FUNCTION_BLOCK SchieberControl (* Basic FB with Schieber ECC *)
  (* Standard: 61499-2; Description: Copyright (c) 2025 HR Agrartechnik GmbH This program and the accompanying materials are made available under the terms of the Eclipse Public License 2.0 which is available at https://www.eclipse.org/legal/epl-2.0/ SPDX-License-Identifier: EPL-2.0 *)
  (* Version 1.0, 2025-06-03, Franz Höpfinger, HR Agrartechnik GmbH *)
  IMPORT Schieber::AufZu::STATES;
  IMPORT Schieber::AufZu::START;
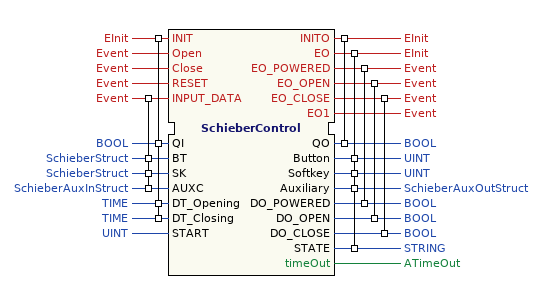
  EVENT_INPUT
    INIT : EInit WITH QI, DT_Opening, DT_Closing; (* Set all Values. Initialization Request. De-Init is not  fully supported. *)
    Open; (* Open *)
    Close; (* Close *)
    RESET; (* Reset to unknown State *)
    INPUT_DATA WITH BT, SK, AUXC;
  END_EVENT
  EVENT_OUTPUT
    INITO : EInit WITH QO; (* All Values have been Set. Initialization Confirm. *)
    EO : EInit WITH Button, Softkey, Auxiliary, STATE;
    EO_POWERED WITH DO_POWERED; (* Actuate "Open" Valve for Pneumatic *)
    EO_OPEN WITH DO_OPEN; (* Actuate "Open" Valve *)
    EO_CLOSE WITH DO_CLOSE; (* Actuate "Close" Valve *)
    EO1;
  END_EVENT
  VAR_INPUT
    QI : BOOL; (* Input event qualifier *)
    BT : SchieberStruct; (* Button *)
    SK : SchieberStruct; (* SoftKey *)
    AUXC : SchieberAuxInStruct; (* Auxiliary Control *)
    DT_Opening : TIME; (* TIME Setting *)
    DT_Closing : TIME; (* TIME Setting *)
    START : UINT := START::STARTUnknown;
  END_VAR
  VAR_OUTPUT
    QO : BOOL; (* Output event qualifier *)
    Button : UINT; (* Button Out *)
    Softkey : UINT; (* Softkey Out *)
    Auxiliary : SchieberAuxOutStruct; (* Auxiliary Control Out *)
    DO_POWERED : BOOL; (* Actuate "Open" Valve for Pneumatic *)
    DO_OPEN : BOOL; (* Actuate "Open" Valve *)
    DO_CLOSE : BOOL; (* Actuate "Close" Valve *)
    STATE : STRING;
  END_VAR
  PLUGS
    timeOut : ATimeOut; (* timeOut Adapter *)
  END_PLUGS
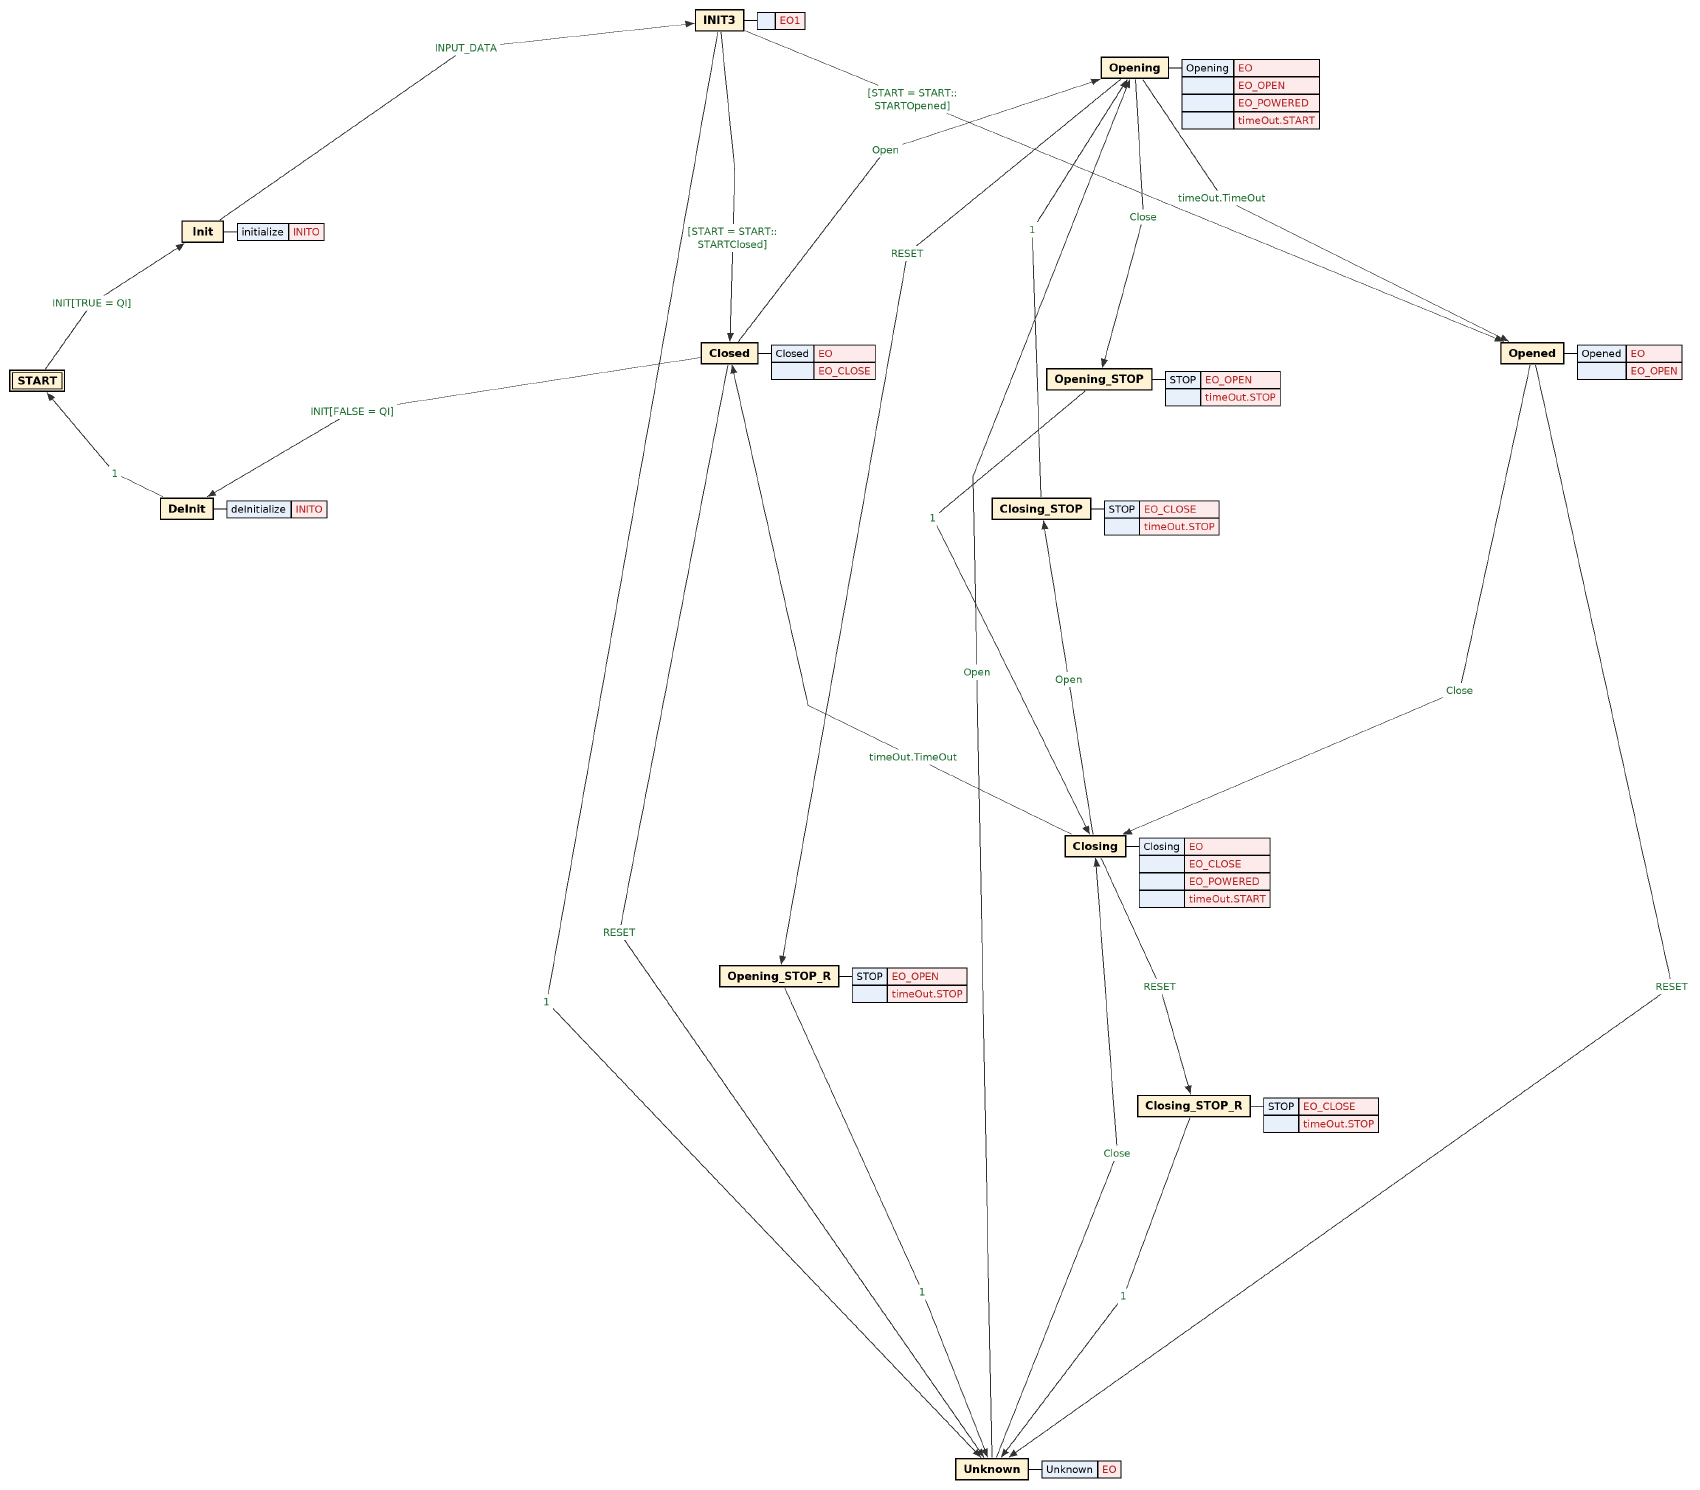
  EC_STATES
    START; (* Initial State *)
    Init : initialize -> INITO; (* Initialization *)
    Closed : Closed -> EO, -> EO_CLOSE;
    DeInit : deInitialize -> INITO;
    Opened : Opened -> EO, -> EO_OPEN;
    Closing : Closing -> EO, -> EO_CLOSE, -> EO_POWERED, -> timeOut.START;
    Opening : Opening -> EO, -> EO_OPEN, -> EO_POWERED, -> timeOut.START;
    Opening_STOP : STOP -> EO_OPEN, -> timeOut.STOP;
    Closing_STOP : STOP -> EO_CLOSE, -> timeOut.STOP;
    Unknown : Unknown -> EO;
    Opening_STOP_R : STOP -> EO_OPEN, -> timeOut.STOP;
    Closing_STOP_R : STOP -> EO_CLOSE, -> timeOut.STOP;
    INIT3 : -> EO1;
  END_STATES
  EC_TRANSITIONS
    START TO Init := INIT[TRUE = QI];
    DeInit TO START := 1;
    Closed TO Opening := Open;
    Closed TO DeInit := INIT[FALSE = QI];
    Opening TO Opened := timeOut.TimeOut;
    Opened TO Closing := Close;
    Closing TO Closed := timeOut.TimeOut;
    Opening TO Opening_STOP := Close;
    Closing TO Closing_STOP := Open;
    Opening_STOP TO Closing := 1;
    Closing_STOP TO Opening := 1;
    Opened TO Unknown := RESET;
    Closed TO Unknown := RESET;
    Opening TO Opening_STOP_R := RESET;
    Closing TO Closing_STOP_R := RESET;
    Opening_STOP_R TO Unknown := 1;
    Closing_STOP_R TO Unknown := 1;
    Unknown TO Opening := Open;
    Unknown TO Closing := Close;
    INIT3 TO Closed := [START = START::STARTClosed];
    Init TO INIT3 := INPUT_DATA;
    INIT3 TO Opened := [START = START::STARTOpened];
    INIT3 TO Unknown := 1;
  END_TRANSITIONS
  ALGORITHM initialize IN ST:
QO := QI;
  END_ALGORITHM
  ALGORITHM deInitialize IN ST:
QO := BOOL#FALSE;
  END_ALGORITHM
  ALGORITHM Closed IN ST:
STATE := STATES::Closed;
Softkey := SK.Closed;
Button := BT.Closed;
Auxiliary.Picture := AUXC.Picture.Closed;
Auxiliary.u8Colour := AUXC.u8Colour.Closed;
DO_POWERED := BOOL#FALSE;
DO_OPEN := BOOL#FALSE;
DO_CLOSE := BOOL#FALSE;
  END_ALGORITHM
  ALGORITHM Opening IN ST:
STATE := STATES::Opening;
Softkey := SK.Opening;
Button := BT.Opening;
Auxiliary.Picture := AUXC.Picture.Opening;
Auxiliary.u8Colour := AUXC.u8Colour.Opening;
timeOut.DT := DT_Opening;
DO_POWERED := BOOL#TRUE;
DO_OPEN := BOOL#TRUE;
DO_CLOSE := BOOL#FALSE;
  END_ALGORITHM
  ALGORITHM Opened IN ST:
STATE := STATES::Opened;
Softkey := SK.Opened;
Button := BT.Opened;
Auxiliary.Picture := AUXC.Picture.Opened;
Auxiliary.u8Colour := AUXC.u8Colour.Opened;
DO_POWERED := BOOL#TRUE;
DO_OPEN := BOOL#FALSE;
DO_CLOSE := BOOL#FALSE;
  END_ALGORITHM
  ALGORITHM Closing IN ST:
STATE := STATES::Closing;
Softkey := SK.Closing;
Button := BT.Closing;
Auxiliary.Picture := AUXC.Picture.Closing;
Auxiliary.u8Colour := AUXC.u8Colour.Closing;
timeOut.DT := DT_Closing;
DO_POWERED := BOOL#FALSE;
DO_OPEN := BOOL#FALSE;
DO_CLOSE := BOOL#TRUE;
  END_ALGORITHM
  ALGORITHM STOP IN ST:
// Powered_unchanged
DO_OPEN := BOOL#FALSE;
DO_CLOSE := BOOL#FALSE;
  END_ALGORITHM
  ALGORITHM Unknown IN ST:
STATE := STATES::Unknown;
Softkey := SK.Unknown;
Button := BT.Unknown;
Auxiliary.Picture := AUXC.Picture.Unknown;
Auxiliary.u8Colour := AUXC.u8Colour.Unknown;
DO_POWERED := BOOL#FALSE;
DO_OPEN := BOOL#FALSE;
DO_CLOSE := BOOL#FALSE;
  END_ALGORITHM
END_FUNCTION_BLOCK
